TYPE ColdRecyclingParameters :
STRUCT
	EN: BOOL := FALSE;
	Offset: LREAL := -2; // Cold recylcing offset (normally negative)
	Hysteresis: lreal := 0.5;
END_STRUCT
END_TYPE

(* stored: Version 1.1.0.1, ProductVersion 3.1.4024.6
   DUT ColdRecyclingParameters: Id {f6de2867-5c0c-4afd-a856-dd48289dbad4} *)
